ABB RobotStudio station: 实验二.rspag

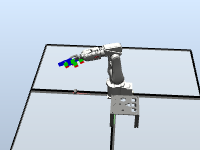
--- station ---
Station PartC (saved by RobotStudio 6.8.8148.134)
Controller System2
  mechanical unit ROB_1: IRB120_3_58__01, 6 joints, base frame (0, 0, 0) mm
Layout (positions relative to the parent item):
  - IRB120_3_58__01 [mechanism, from Robots\IRB120_3_58_G_01.rslib] at (0, 0, 0) mm; joint values [0.3383, 0.1087, -0.0614, -0.0001, 0.2519, 0.0387] (rad or m)
  - SmartComponent_1 [smart component] at (380.22, 133.79, 592.82) mm, rotated rx 172.87 ry 72.72 rz -168.08 deg
      signals: DI GET, DO FINISH
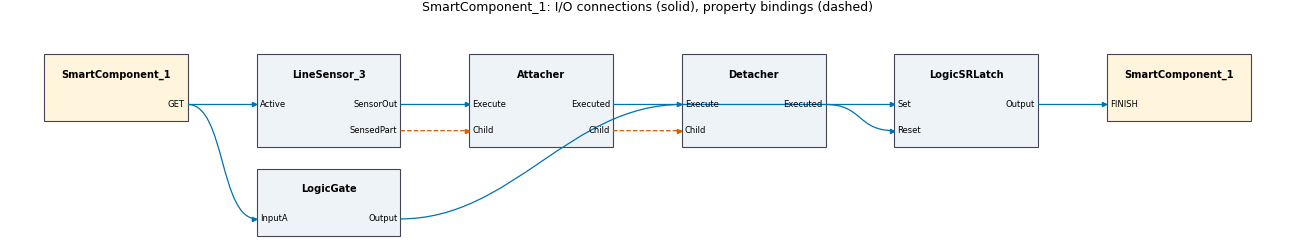
      connections:
        SmartComponent_1.GET -> LineSensor_3.Active
        SmartComponent_1.GET -> LogicGate.InputA
        LineSensor_3.SensorOut -> Attacher.Execute
        LogicGate.Output -> Detacher.Execute
        Attacher.Executed -> LogicSRLatch.Set
        Detacher.Executed -> LogicSRLatch.Reset
        LogicSRLatch.Output -> SmartComponent_1.FINISH
        LineSensor_3.SensedPart => Attacher.Child
        Attacher.Child => Detacher.Child
    - LineSensor_3 [smart component, from Components\LineSensor.rslib] at (-22.5, 0, 83.55) mm
        properties: Start=[0.0150000000000009 -0.000761999999999613 0.00306099999999904]; End=[-0.0249959999999991 0.00111800000000039 0.00431999999999905]; Radius=0.005; SensedPart=TCP-练习笔; SensedPoint=[-0.0910465469360352 0.454929412841797 0.202439468383789]
      - _sensorPart_ [part]
    - Attacher [smart component, from Components\Attacher.rslib]
        properties: Parent=SmartComponent_1; Flange=0; Child=TCP-练习笔; Mount=false; Offset=[0 0 0]; Orientation=[0 0 0]
    - Detacher [smart component, from Components\Detacher.rslib]
        properties: Child=TCP-练习笔; KeepPosition=true
    - LogicGate [smart component, from Components\LogicGate.rslib]
        properties: Operator=NOT; Delay=0
    - LogicSRLatch [smart component, from Components\LogicSRLatch.rslib]
    - My_Mechanism [mechanism] at (0, 0, 0) mm; joint values [0.01] (rad or m)
        TCP tool1 at (15.5, 0, 69.3) mm
        TCP tool2 at (-22.5, 0, 83.55) mm
        TCP tool3 at (-22.5, 0, 160.55) mm
        links: L1, L2
  - 部件_2 [part] at (0, 0, 23.06) mm
  - TCP_Table [part]
  - TCP-练习笔 [part] at (0, 0, 0.59) mm
  - 框架_1 [frame] at (15.5, 0, 69.3) mm
  - 框架_2 [frame] at (-22.5, 0, 83.55) mm
  - 框架_3 [frame] at (-22.5, 0, 160.55) mm
Attachment: My_Mechanism is attached to IRB120_3_58__01 / Link6
Attachment: SmartComponent_1 is attached to IRB120_3_58__01 / Link6
Attachment: LineSensor_3 is attached to My_Mechanism / L1
EventTableEntry 2443: Group=, Trigger=DO_007 2444, Actions=[EventTableActionMechanicalPose 2445], Comment=, ActivationMode=2, Cyclic=false
EventTableTriggerIO 2444: IOValue=[1], IRC5Controller=? -1, Operator=0, SignalSource=System2 2451
EventTableActionMechanicalPose 2445: VirtualSignal=, Mechanism=My_Mechanism 980, ToPoseName=SyncPosition, VirtualSignalValue=[1]
EventTableEntry 2446: Group=, Trigger=DO_007 2447, Actions=[EventTableActionMechanicalPose 2448], Comment=, ActivationMode=2, Cyclic=false
EventTableTriggerIO 2447: IOValue=[0], IRC5Controller=? -1, Operator=0, SignalSource=System2 2451
EventTableActionMechanicalPose 2448: VirtualSignal=, Mechanism=My_Mechanism 980, ToPoseName=HomePosition, VirtualSignalValue=[1]
Station logic (signal -> signal, property => property):
  System2.DO_007 -> SmartComponent_1.GET
Targets, tools, work objects and paths stored in the station and not in the controller backup, written as RAPID:
! task T_ROB1
MODULE CalibData
  PERS tooldata tool1:=[TRUE,[[15.5,0,69.3],[1,0,0,0]],[1,[0,0,1],[1,0,0,0],0,0,0]];
  PERS tooldata tool2:=[TRUE,[[-22.5,0,83.554],[1,0,0,0]],[1,[0,0,1],[1,0,0,0],0,0,0]];
  PERS tooldata tool3:=[TRUE,[[-22.5,0,160.554],[1,0,0,0]],[1,[0,0,1],[1,0,0,0],0,0,0]];
  PERS tooldata Tooldata_4:=[TRUE,[[15.5,0,69.3],[1,0,0,0]],[1,[0,0,1],[1,0,0,0],0,0,0]];
  PERS tooldata Tooldata_5:=[TRUE,[[-22.5,0,83.554],[1,0,0,0]],[1,[0,0,1],[1,0,0,0],0,0,0]];
  PERS tooldata Tooldata_6:=[TRUE,[[-22.5,0,160.554],[1,0,0,0]],[1,[0,0,1],[1,0,0,0],0,0,0]];
ENDMODULE


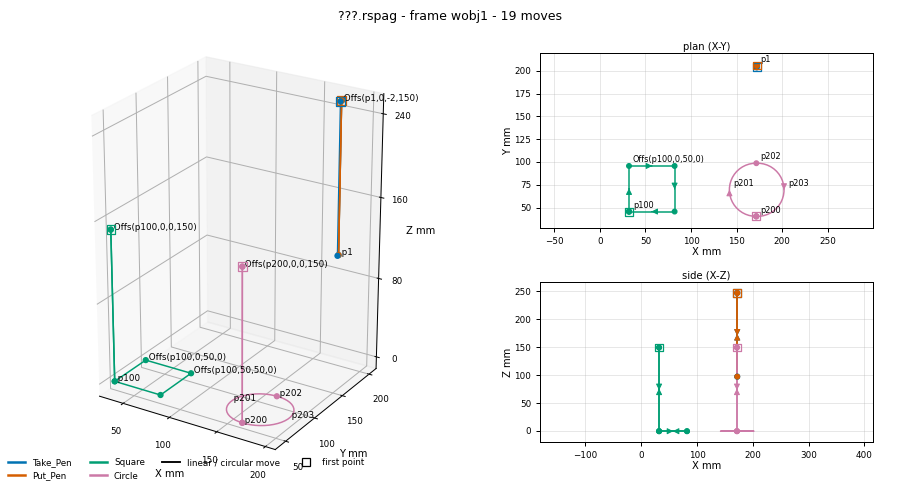
[picture p0: tool path of 实验二.rspag in frame wobj1, 19 of 21 moves have a stored position in this frame; points joined in program order, loops and branches not executed]
--- Backups/System2/RAPID/TASK1/PROGMOD/Module1.mod ---
MODULE Module1
	TASK PERS loaddata load1:=[1,[0,0,50],[1,0,0,0],0,0,0];
	CONST robtarget p1:=[[172.01,205.77,97.31],[0.00112688,-0.706761,0.707451,0.00098463],[1,-1,0,0],[9E+9,9E+9,9E+9,9E+9,9E+9,9E+9]];
	CONST robtarget p11:=[[263.58,61.16,366.17],[0.000305777,-0.706762,0.707451,0.000164551],[1,0,0,0],[9E+9,9E+9,9E+9,9E+9,9E+9,9E+9]];
	CONST robtarget p21:=[[172.01,205.77,97.31],[0.00112688,-0.706761,0.707451,0.00098463],[1,-1,0,0],[9E+9,9E+9,9E+9,9E+9,9E+9,9E+9]];
	CONST robtarget p100:=[[31.94,45.61,-0.49],[0.00223608,-0.000486235,-0.999989,-0.00403198],[1,-1,0,0],[9E+9,9E+9,9E+9,9E+9,9E+9,9E+9]];
	CONST robtarget p200:=[[171.47,40.35,-0.47],[0.00223616,-0.000486939,-0.999989,-0.00403224],[1,0,0,0],[9E+9,9E+9,9E+9,9E+9,9E+9,9E+9]];
	CONST robtarget p220:=[[172.01,205.77,97.31],[0.00112688,-0.706761,0.707451,0.00098463],[1,-1,0,0],[9E+9,9E+9,9E+9,9E+9,9E+9,9E+9]];
	CONST robtarget p210:=[[172.01,205.77,97.31],[0.00112688,-0.706761,0.707451,0.00098463],[1,-1,0,0],[9E+9,9E+9,9E+9,9E+9,9E+9,9E+9]];
	CONST robtarget p201:=[[142.00,69.14,-0.45],[0.00223618,-0.000487262,-0.999989,-0.00403234],[1,0,0,0],[9E+9,9E+9,9E+9,9E+9,9E+9,9E+9]];
	CONST robtarget p202:=[[171.58,98.63,-0.43],[0.00223622,-0.000487166,-0.999989,-0.0040324],[1,0,0,0],[9E+9,9E+9,9E+9,9E+9,9E+9,9E+9]];
	CONST robtarget p203:=[[201.97,69.09,-0.44],[0.00223617,-0.000487189,-0.999989,-0.00403229],[1,0,0,0],[9E+9,9E+9,9E+9,9E+9,9E+9,9E+9]];
	CONST robtarget p213:=[[172.01,205.77,97.31],[0.00112688,-0.706761,0.707451,0.00098463],[1,-1,0,0],[9E+9,9E+9,9E+9,9E+9,9E+9,9E+9]];
    !***********************************************************
    !
    ! Module:  Module1
    !
    ! Description:
    !   <Insert description here>
    !
    ! Author: He
    !
    ! Version: 1.0
    !
    !***********************************************************


    !***********************************************************
    !
    ! Procedure main
    !
    !   This is the entry point of your program
    !
    !***********************************************************
    PROC main()
        Initialize;
        Take_Pen;
        Square;
        Circle;
        Put_Pen;
    ENDPROC
	PROC Initialize()
		AccSet 100, 100;
		VelSet 100, 300;
		MoveAbsJ [[0,0,0,0,0,0],[9E+9,9E+9,9E+9,9E+9,9E+9,9E+9]]\NoEOffs, v100, z50, tool0;
		Reset DO_007;
		MoveAbsJ [[90,0,0,0,90,0],[9E+9,9E+9,9E+9,9E+9,9E+9,9E+9]]\NoEOffs, v100, z50, tool0;
	ENDPROC
	PROC Take_Pen()
		MoveJ Offs(p1,0,-2,150), v100, z50, tool0\WObj:=wobj1;
		MoveL Offs(p1,0,-2,0), v50, fine, tool0\WObj:=wobj1;
		MoveL p1, v50, fine, tool0\WObj:=wobj1;
		Set DO_007;
		WaitTime 1;
		MoveL Offs(p1,0,0,150), v100, z50, tool0\WObj:=wobj1;
	ENDPROC
	PROC Put_Pen()
		MoveJ Offs(p1,0,0,150), v100, z50, tool0\WObj:=wobj1;
		MoveL p1, v50, fine, tool0\WObj:=wobj1;
		Reset DO_007;
		WaitTime 1;
		MoveL Offs(p1,0,0,150), v100, z50, tool0\WObj:=wobj1;
	ENDPROC
	PROC Square()
		MoveJ Offs(p100,0,0,150), v100, z50, tool_pen\WObj:=wobj1;
		MoveL p100, v50, fine, tool_pen\WObj:=wobj1;
		MoveL Offs(p100,0,50,0), v100, z50, tool_pen\WObj:=wobj1;
		MoveL Offs(p100,50,50,0), v100, z50, tool_pen\WObj:=wobj1;
		MoveL Offs(p100,50,0,0), v100, z50, tool_pen\WObj:=wobj1;
		MoveL p100, v100, fine, tool_pen\WObj:=wobj1;
		MoveL Offs(p100,0,0,150), v100, z50, tool_pen\WObj:=wobj1;
	ENDPROC
	PROC Circle()
		MoveJ Offs(p200,0,0,150), v100, z50, tool_pen\WObj:=wobj1;
		MoveL p200, v50, fine, tool_pen\WObj:=wobj1;
		MoveC p201, p202, v100, z50, tool_pen\WObj:=wobj1;
		MoveC p203, p200, v100, fine, tool_pen\WObj:=wobj1;
		MoveL Offs(p200,0,0,150), v100, z10, tool_pen\WObj:=wobj1;
	ENDPROC
ENDMODULE

--- Backups/System2/SYSPAR/EIO.cfg ---
EIO:CFG_1.0:6:1::
#
INDUSTRIAL_NETWORK:

      -Name "DeviceNet" -Label "DeviceNet Master/Slave Network" -Address "2"
#
DEVICENET_DEVICE:

      -Name "d652" -VendorName "ABB Robotics" -ProductName "24 VDC I/O Device"\
      -Label "DSQC 652 24 VDC I/O Device" -Address 10 -ProductCode 26\
      -DeviceType 7 -ConnectionType "COS" -OutputSize 2 -InputSize 2
#
DEVICENET_INTERNAL_DEVICE:

      -Name "DN_Internal_Device" -VendorName "ABB Robotics"\
      -ProductName "DeviceNet Internal Slave Device"
#
EIO_SIGNAL:

      -Name "DO_007" -SignalType "DO" -Device "d652" -DeviceMap "7"
